{attribute 'qualified_only'}
{attribute 'strict'}
TYPE eTcoComponentTests : 
(
    GetSignalInfo := 100
);
END_TYPE

(* stored: Version 1.1.0.1
   DUT eTcoComponentTests: Id {75192e0b-d303-092f-2908-00d3094eab29} *)
